// TwinCAT 3 PLC project Samples
// ProgramVersion: 3.1.4023.0
// libraries:
//   Tc2_Standard, * (Beckhoff Automation GmbH)
//   Tc2_System, * (Beckhoff Automation GmbH)
//   Tc3_Module, * (Beckhoff Automation GmbH)
// project tree:
//   DUTs/ PLCStruct.TcDUT
//   GVLs/ GVL.TcGVL
//   / PlcTask.TcTTO
//   POUs/ MAIN.TcPOU
// real-time tasks:
//   TASK PlcTask: cycle T#10ms, priority 20, ADS port 350

CONFIGURATION Samples
    RESOURCE PLC ON TwinCAT3
        TASK PlcTask(INTERVAL := T#10ms, PRIORITY := 20);
        PROGRAM MAIN WITH PlcTask : MAIN;
    END_RESOURCE
END_CONFIGURATION

// ---- DUTs/PLCStruct.TcDUT
TYPE PLCStruct :
STRUCT
    intVal		AT	%MB0	: 	INT;
    dintVal		AT	%MB2	: 	DINT;
    sintVal		AT	%MB6	: 	SINT;
    lrealVal	AT	%MB7	: 	LREAL;
    realVal		AT	%MB15	: 	REAL;
END_STRUCT
END_TYPE

// ---- GVLs/GVL.TcGVL
VAR_GLOBAL
	// Sample 05
	PLCVarBYTE       AT %MB500    : BYTE;
	PLCVarWORD       AT %MB502    : WORD;
	PLCVarDWORD	     AT %MB504    : DWORD;
	PLCVarBOOL       AT %MX508.0  : BOOL;
	PLCVarINT        AT %MB510    : INT;
	PLCVarUINT       AT %MB512    : UINT;
	PLCVarSINT       AT %MB514    : SINT;
	PLCVarUSINT      AT %MB516    : USINT;
	PLCVarDINT       AT %MB520    : DINT;
	PLCVarUDINT      AT %MB524    : UDINT := 1234;
	PLCVarREAL       AT %MB528    : REAL;
	PLCVarLREAL      AT %MB536    : LREAL;
	PLCVarUDINTArray	          : ARRAY[0..5] OF UDINT :=[ 5,4,3,2,1,0];

	// Sample 11
	SPSVar1                       : DWORD;
	SPSVar2                       : DWORD;
	SPSVar3                       : DWORD;
	SPSVar4                       : DWORD;

	// Sample 12
	bVar01           AT %QX1200.0 : BOOL;
	bVar02           AT %QX1200.1 : BOOL;
END_VAR

// ---- POUs/MAIN.TcPOU
PROGRAM MAIN
VAR
	// Sample 02
	PLCVar2                : DWORD;
	TP_2                   : TP;
	TOGGEL2                : BOOL;
	
	// Sample 03
 	PLCVar3   AT %MB300    : ARRAY [0..99] OF INT;
	Index                  : BYTE;
	
	// Sample 04
	PLCVar4   AT %MB400    : PLCStruct;
	
	// Sample 06
	PLCVar6   AT %MD600    : DWORD;
	
	// Sample 07 & Sample 08 & Sample 09
	PLCVar    AT %MD0      : DWORD;
	TP_1                   : TP;
	TOGGEL                 : BOOL;
	
	// Sample 12
	i                      : INT;
	
	// Sample 13
	uintValue AT %MB1300   : UINT := 54321;
	boolValue AT %MX1308.0 : BOOL := TRUE;
	dintValue AT %MB1316   : DINT := -12345678;
END_VAR

// Sample 02
TOGGEL2 := NOT TOGGEL;
TP_2( IN := TOGGEL2, PT := T#1S);
IF (TP_2.Q = 0) THEN
	PLCVar2 := PLCVar2 + 1;
END_IF

// Sample 03
FOR Index := 0 TO 99 DO
  PLCVar3[Index] := UINT_TO_INT(3500 + INDEX);
END_FOR

// Sample 07 & Sample 08 & Sample 09
TOGGEL := NOT TOGGEL;
TP_1(IN := TOGGEL, PT := T#1S);
IF (TP_1.Q = 0) THEN
	PLCVar := PLCVar + 1;
END_IF

// Sample 12
i := i+1;
IF i >= 0 THEN
	bVar01 := TRUE;
	bVar02 := FALSE;
END_IF
IF i >= 100 THEN
	bVar01 := FALSE;
	bVar02 := TRUE;
END_IF
IF i >= 200 THEN
	i := 0;
END_IF

END_PROGRAM
